FUNCTION Rejection_Codes_Function : STRING
VAR_INPUT
	Fixture_Code	: INT;
END_VAR
VAR	

END_VAR

IF Fixture_Code = 0 OR Fixture_Code >151 THEN
	Rejection_Codes_Function:=' NA ';
END_IF
IF Fixture_Code = 21 THEN
	Rejection_Codes_Function:='  OP20';
END_IF
IF Fixture_Code = 31 THEN
	Rejection_Codes_Function:='  OP30';
END_IF
IF Fixture_Code = 41 THEN
	Rejection_Codes_Function:='  OP40';
END_IF
IF Fixture_Code = 51 THEN
	Rejection_Codes_Function:='  OP50';
END_IF
IF Fixture_Code = 61 THEN
	Rejection_Codes_Function:='  OP60';
END_IF
IF Fixture_Code = 71 THEN
	Rejection_Codes_Function:='  OP70';
END_IF
IF Fixture_Code = 81 THEN
	Rejection_Codes_Function:='  OP80';
END_IF
IF Fixture_Code = 91 THEN
	Rejection_Codes_Function:='  OP90';
END_IF
IF Fixture_Code = 111 THEN
	Rejection_Codes_Function:='  OP110';
END_IF
IF Fixture_Code = 121 THEN
	Rejection_Codes_Function:='  OP120';
END_IF
IF Fixture_Code = 131 THEN
	Rejection_Codes_Function:='  OP130';
END_IF
IF Fixture_Code = 141 THEN
	Rejection_Codes_Function:='  OP140';
END_IF
IF Fixture_Code = 151 THEN
	Rejection_Codes_Function:='  OP150-V';
END_IF

END_FUNCTION

(* stored: Version 1.1.0.1, ProductVersion 3.1.4024.11
   POU Rejection_Codes_Function: Id {2bcbdead-ab76-4953-9d91-d1aa69abb9a0}, SpecialFunc None *)
